INTERFACE ITF_OutputDevice

METHOD WriteControlOutputs : BOOL
VAR_INPUT
END_VAR
END_METHOD

END_INTERFACE

(* stored: Version 1.1.0.1, ProductVersion 3.1.4024.12
   Itf ITF_OutputDevice: Id {cc4b4379-1174-4f89-9109-bb7f8802e218}
   Method WriteControlOutputs: Id {de5ed4ab-40a0-408c-8931-6b35227c5f3b} *)
